{attribute 'qualified_only'}
VAR_GLOBAL CONSTANT
  MaxJsonKeyLength : INT := 31;
  MaxJsonAssignments : INT := 200;
END_VAR

(* stored: Version 1.1.0.1, ProductVersion 3.1.4024.12
   GVL ParameterList: Id {64e570dd-c626-47da-b2c7-1e2c8664fa9d}, ParameterList True *)
